{attribute 'qualified_only'}
{attribute 'strict'}
{attribute 'to_string'}
TYPE E_Mode :
(
	Tune 	:=0,
	Run		:=1
);
END_TYPE

(* stored: Version 1.1.0.1, ProductVersion 3.1.4024.12
   EnumerationTextList E_Mode: Id {9a2d9ae3-94e7-413c-9910-89140bbf1d75} *)
